TYPE ST_DischargeStatus :
STRUCT
    eStep                   : E_DischargeState;
    bDone                   : BOOL;
    bAutoTakeOver           : BOOL;
    bWaitingForBagChange    : BOOL;
    sDiag                   : T_MaxString;
END_STRUCT
END_TYPE

(* stored: Version 1.1.0.1, ProductVersion 3.1.4024.16
   DUT ST_DischargeStatus: Id {250fda01-126d-4c5b-87e2-ca4da10811ea} *)
